(* IEC 61131-3 sources: AutomationBullShit/RevolvingDoor_poST, 5 files *)

(* ---- GVL.st ---- *)
{attribute 'qualified_only' := 'false'}
VAR_GLOBAL
    (* Presence sensors *)
    presenceSideA           : BOOL;
    presenceSideB           : BOOL;
    (* Presence triggers - visualization writes here *)
    presenceTriggerA        : BOOL;
    presenceTriggerB        : BOOL;
    (* Partition pressure sensor *)
    partitionPressure       : BOOL;
    (* Manual rotation buttons *)
    rotateForwardButton     : BOOL;
    rotateBackwardButton    : BOOL;
    (* Rotation direction: FALSE=counter-clockwise (default), TRUE=clockwise *)
    rotationClockwise       : BOOL;
    (* Door angle sensor *)
    doorAngle               : REAL;
(* Rotation status *)
    isRotating              : BOOL;
    (* Motor control *)
    motorOn                 : BOOL;
    rotationForward         : BOOL;
    (* Motor enable switch *)
    motorEnable             : BOOL := TRUE;
    (* Emergency stop *)
    emergencyStop           : BOOL;
    (* Traffic lights *)
    lightSideA              : BOOL;
    lightSideB              : BOOL;
END_VAR

(* ---- Controller_DECL.st ---- *)
PROGRAM Controller
VAR CONSTANT
    ROTATION_TIME   : INT := 100;
    REVERSE_TICKS   : INT := 50;    (* 5 degrees at ROTATION_SPEED=0.1 *)
END_VAR
VAR
    (* MainControl state: 0=idle, 1=rotating, 2=manualRotation, 3=pressure *)
    mainState               : INT := 0;
    timer                   : INT := 0;
    manualActive            : BOOL := FALSE;
    manualDirectionForward  : BOOL := TRUE;
    (* Pressure sub-process: 0=released, 1=reversing, 2=stopped *)
    pauseState              : INT := 0;
    reverseCounter          : INT := 0;
END_VAR

(* ---- Controller_IMPL.st ---- *)
(* Emergency stop - disable motor *)
IF GVL.emergencyStop THEN
    GVL.motorEnable := FALSE;
END_IF

(* Motor disabled - immediate stop, reset to idle *)
IF NOT GVL.motorEnable THEN
    GVL.motorOn := FALSE;
    GVL.rotationForward := NOT GVL.rotationClockwise;
    GVL.lightSideA := FALSE;
    GVL.lightSideB := FALSE;
	GVL.presenceSideA := FALSE;
    GVL.presenceSideB := FALSE;
    manualActive := FALSE;
    timer := 0;
    pauseState := 0;
    mainState := 0;
ELSE

CASE mainState OF

0: (* idle *)
    GVL.lightSideA := TRUE;
    GVL.lightSideB := TRUE;
    IF GVL.rotateForwardButton AND NOT GVL.rotateBackwardButton AND NOT GVL.partitionPressure THEN
        manualActive := TRUE;
        manualDirectionForward := TRUE;
        GVL.motorOn := TRUE;
        GVL.rotationForward := NOT GVL.rotationClockwise;
        GVL.lightSideA := TRUE;
        GVL.lightSideB := TRUE;
        mainState := 2;

    ELSIF GVL.rotateBackwardButton AND NOT GVL.rotateForwardButton AND NOT GVL.partitionPressure THEN
        manualActive := TRUE;
        manualDirectionForward := FALSE;
        GVL.motorOn := TRUE;
        GVL.rotationForward := GVL.rotationClockwise;
        GVL.lightSideA := TRUE;
        GVL.lightSideB := TRUE;
        mainState := 2;

    ELSIF (GVL.presenceSideA OR GVL.presenceSideB) AND NOT GVL.partitionPressure THEN
        manualActive := FALSE;
        manualDirectionForward := TRUE;
        GVL.motorOn := TRUE;
        GVL.rotationForward := NOT GVL.rotationClockwise;
        GVL.lightSideA := TRUE;
        GVL.lightSideB := TRUE;
        timer := ROTATION_TIME;
        mainState := 1;
    END_IF

1: (* rotating *)
    IF (GVL.presenceSideA OR GVL.presenceSideB) THEN
        timer := ROTATION_TIME;
    END_IF

    IF GVL.partitionPressure THEN
        GVL.motorOn := FALSE;
        GVL.rotationForward := NOT GVL.rotationForward;
        GVL.lightSideA := FALSE;
        GVL.lightSideB := FALSE;
        reverseCounter := REVERSE_TICKS;
        pauseState := 1;
        mainState := 3;
    ELSIF NOT (GVL.presenceSideA OR GVL.presenceSideB) THEN
        timer := timer - 1;
    END_IF

    IF timer <= 0 AND mainState = 1 THEN
        GVL.motorOn := FALSE;
        GVL.rotationForward := NOT GVL.rotationClockwise;
        GVL.lightSideA := TRUE;
        GVL.lightSideB := TRUE;
        mainState := 0;
    END_IF

2: (* manualRotation *)
    IF GVL.partitionPressure THEN
        GVL.motorOn := FALSE;
        GVL.rotationForward := NOT GVL.rotationForward;
        GVL.lightSideA := FALSE;
        GVL.lightSideB := FALSE;
        reverseCounter := REVERSE_TICKS;
        pauseState := 1;
        mainState := 3;

    ELSIF GVL.rotateForwardButton AND GVL.rotateBackwardButton THEN
        GVL.motorOn := FALSE;
        GVL.rotationForward := NOT GVL.rotationClockwise;
        GVL.lightSideA := TRUE;
        GVL.lightSideB := TRUE;
        manualActive := FALSE;
        mainState := 0;

    ELSIF manualDirectionForward AND GVL.rotateForwardButton THEN
        GVL.motorOn := TRUE;
        GVL.rotationForward := NOT GVL.rotationClockwise;
        GVL.lightSideA := TRUE;
        GVL.lightSideB := TRUE;

    ELSIF (NOT manualDirectionForward) AND GVL.rotateBackwardButton THEN
        GVL.motorOn := TRUE;
        GVL.rotationForward := GVL.rotationClockwise;
        GVL.lightSideA := TRUE;
        GVL.lightSideB := TRUE;

    ELSE
        GVL.motorOn := FALSE;
        GVL.rotationForward := NOT GVL.rotationClockwise;
        GVL.lightSideA := TRUE;
        GVL.lightSideB := TRUE;
        manualActive := FALSE;
        mainState := 0;
    END_IF

3: (* pressure reaction *)
    IF pauseState = 1 THEN
        (* Reversing 5 degrees *)
        GVL.motorOn := TRUE;
        reverseCounter := reverseCounter - 1;
        IF reverseCounter <= 0 THEN
            GVL.motorOn := FALSE;
            pauseState := 2;
        END_IF
    END_IF

    IF pauseState = 2 THEN
        (* Stopped until pressure released *)
        GVL.motorOn := FALSE;
        IF NOT GVL.partitionPressure THEN
            pauseState := 0;
        END_IF
    END_IF

    IF pauseState = 0 THEN
        (* Pressure released - resume *)
        IF manualActive THEN
            IF manualDirectionForward AND GVL.rotateForwardButton THEN
                GVL.motorOn := TRUE;
                GVL.rotationForward := NOT GVL.rotationClockwise;
                GVL.lightSideA := TRUE;
                GVL.lightSideB := TRUE;
                mainState := 2;
            ELSIF (NOT manualDirectionForward) AND GVL.rotateBackwardButton THEN
                GVL.motorOn := TRUE;
                GVL.rotationForward := GVL.rotationClockwise;
                GVL.lightSideA := TRUE;
                GVL.lightSideB := TRUE;
                mainState := 2;
            ELSE
                GVL.motorOn := FALSE;
                GVL.rotationForward := NOT GVL.rotationClockwise;
                GVL.lightSideA := TRUE;
                GVL.lightSideB := TRUE;
                manualActive := FALSE;
                mainState := 0;
            END_IF
        ELSIF timer > 0 THEN
            GVL.motorOn := TRUE;
            GVL.rotationForward := NOT GVL.rotationClockwise;
            GVL.lightSideA := TRUE;
            GVL.lightSideB := TRUE;
            mainState := 1;
        ELSE
            GVL.motorOn := FALSE;
            GVL.rotationForward := NOT GVL.rotationClockwise;
            GVL.lightSideA := TRUE;
            GVL.lightSideB := TRUE;
            mainState := 0;
        END_IF
    END_IF

END_CASE

END_IF (* motorEnable / emergencyStop *)

(* ---- Plant_DECL.st ---- *)
PROGRAM Plant
VAR CONSTANT
    ROTATION_SPEED  : REAL := 0.1;
    MAX_ANGLE       : REAL := 360.0;
    PRESENCE_HOLD   : INT := 500;
END_VAR
VAR
    initialized      : BOOL := FALSE;
    presenceTimerA   : INT := 0;
    presenceTimerB   : INT := 0;
END_VAR

(* ---- Plant_IMPL.st ---- *)
IF NOT initialized THEN
    GVL.doorAngle            := 0.0;
    GVL.presenceSideA        := FALSE;
    GVL.presenceSideB        := FALSE;
    GVL.presenceTriggerA     := FALSE;
    GVL.presenceTriggerB     := FALSE;
    presenceTimerA           := 0;
    presenceTimerB           := 0;
    initialized              := TRUE;
END_IF

(* Presence hold - trigger is set by visualization, timer keeps presence active *)
IF GVL.presenceTriggerA THEN
    presenceTimerA := PRESENCE_HOLD;
    GVL.presenceTriggerA := FALSE;
END_IF
GVL.presenceSideA := (presenceTimerA > 0);
IF presenceTimerA > 0 THEN
    presenceTimerA := presenceTimerA - 1;
END_IF

IF GVL.presenceTriggerB THEN
    presenceTimerB := PRESENCE_HOLD;
    GVL.presenceTriggerB := FALSE;
END_IF
GVL.presenceSideB := (presenceTimerB > 0);
IF presenceTimerB > 0 THEN
    presenceTimerB := presenceTimerB - 1;
END_IF

(* MotorSim *)
GVL.isRotating := GVL.motorOn;

(* DoorRotationSim *)
IF GVL.isRotating THEN
    IF GVL.rotationForward THEN
        GVL.doorAngle := GVL.doorAngle - ROTATION_SPEED;
    ELSE
        GVL.doorAngle := GVL.doorAngle + ROTATION_SPEED;
    END_IF
END_IF

IF GVL.doorAngle >= MAX_ANGLE THEN
    GVL.doorAngle := GVL.doorAngle - MAX_ANGLE;
END_IF
IF GVL.doorAngle < 0.0 THEN
    GVL.doorAngle := GVL.doorAngle + MAX_ANGLE;
END_IF
